FUNCTION_BLOCK JackControl (* Composite Function Block Type *)
  (* Standard: 61499-2 *)
  (* Version 0.0, 4/16/2020, prana, nxtControl GmbH, template *)
  PACKAGE Main;
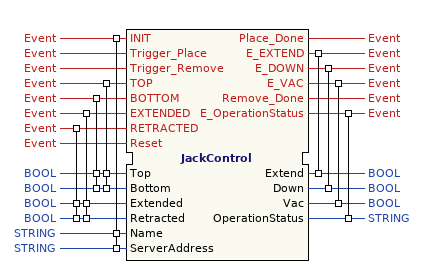
  EVENT_INPUT
    INIT WITH Name, ServerAddress; (* Initialization Request *)
    Trigger_Place;
    Trigger_Remove;
    TOP WITH Top, Bottom; {SET_ATTRIBUTE(Runtime.OPCUA.Access, 2)}
    BOTTOM WITH Bottom, Top; {SET_ATTRIBUTE(Runtime.OPCUA.Access, 2)}
    EXTENDED WITH Extended, Retracted; {SET_ATTRIBUTE(Runtime.OPCUA.Access, 2)}
    RETRACTED WITH Retracted, Extended; {SET_ATTRIBUTE(Runtime.OPCUA.Access, 2)}
    Reset;
  END_EVENT
  EVENT_OUTPUT
    Place_Done;
    E_EXTEND WITH Extend;
    E_DOWN WITH Down;
    E_VAC WITH Vac;
    Remove_Done;
    E_OperationStatus WITH OperationStatus; (* Execution Confirmation *)
  END_EVENT
  VAR_INPUT
    Top : BOOL; {SET_ATTRIBUTE(Runtime.OPCUA.Access, 2)} {SET_ATTRIBUTE(Runtime.OPCUA.WriteTrigger, TOP)}
    Bottom : BOOL; {SET_ATTRIBUTE(Runtime.OPCUA.Access, 2)} {SET_ATTRIBUTE(Runtime.OPCUA.WriteTrigger, BOTTOM)}
    Extended : BOOL; {SET_ATTRIBUTE(Runtime.OPCUA.Access, 2)} {SET_ATTRIBUTE(Runtime.OPCUA.WriteTrigger, EXTENDED)}
    Retracted : BOOL; {SET_ATTRIBUTE(Runtime.OPCUA.Access, 2)} {SET_ATTRIBUTE(Runtime.OPCUA.WriteTrigger, RETRACTED)}
    Name : STRING;
    ServerAddress : STRING;
  END_VAR
  VAR_OUTPUT
    Extend : BOOL; {SET_ATTRIBUTE(Runtime.OPCUA.Access, 2)}
    Down : BOOL; {SET_ATTRIBUTE(Runtime.OPCUA.Access, 2)}
    Vac : BOOL; {SET_ATTRIBUTE(Runtime.OPCUA.Access, 2)}
    OperationStatus : STRING; (* Output event qualifier *)
  END_VAR
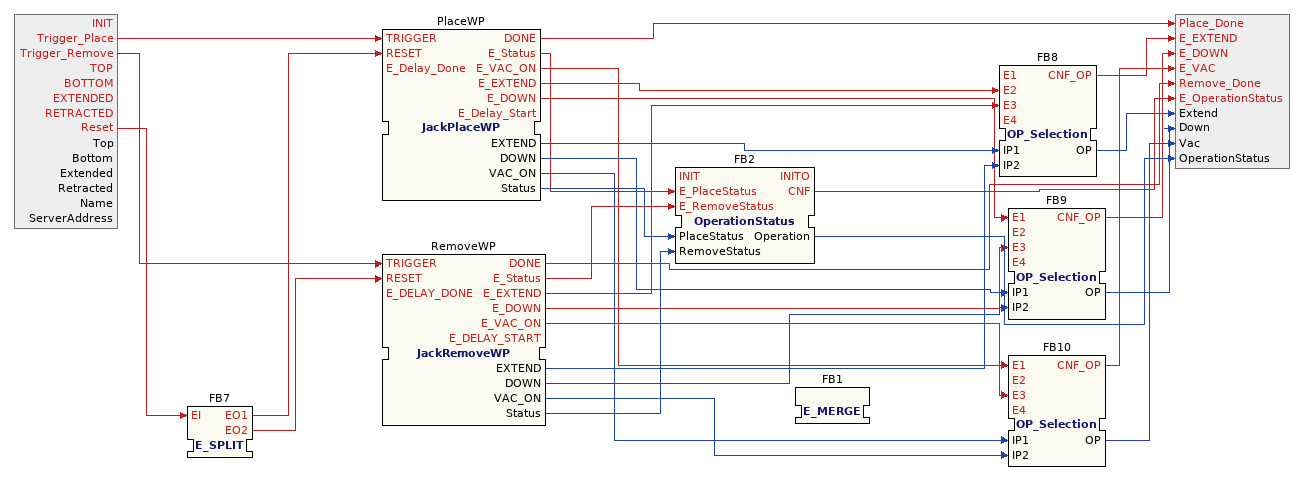
  FBS
    PlaceWP : JackPlaceWP;
    RemoveWP : JackRemoveWP;
    FB7 : E_SPLIT;
    FB8 : OP_Selection;
    FB9 : OP_Selection;
    FB10 : OP_Selection;
    FB1 : E_MERGE;
    FB2 : OperationStatus;
  END_FBS
  EVENT_CONNECTIONS
    Trigger_Place TO PlaceWP.TRIGGER;
    Trigger_Remove TO RemoveWP.TRIGGER;
    Reset TO FB7.EI;
    FB7.EO1 TO PlaceWP.RESET;
    FB7.EO2 TO RemoveWP.RESET;
    FB8.CNF_OP TO E_EXTEND;
    FB9.CNF_OP TO E_DOWN;
    FB10.CNF_OP TO E_VAC;
    RemoveWP.E_VAC_ON TO FB10.E3;
    PlaceWP.E_VAC_ON TO FB10.E1;
    RemoveWP.E_DOWN TO FB9.E3;
    PlaceWP.E_DOWN TO FB9.E1;
    PlaceWP.E_EXTEND TO FB8.E2;
    RemoveWP.E_EXTEND TO FB8.E3;
    PlaceWP.DONE TO Place_Done;
    RemoveWP.DONE TO Remove_Done;
    PlaceWP.E_Status TO FB2.E_PlaceStatus;
    RemoveWP.E_Status TO FB2.E_RemoveStatus;
    FB2.CNF TO E_OperationStatus;
  END_CONNECTIONS
  DATA_CONNECTIONS
    FB8.OP TO Extend;
    FB9.OP TO Down;
    FB10.OP TO Vac;
    RemoveWP.VAC_ON TO FB10.IP2;
    PlaceWP.VAC_ON TO FB10.IP1;
    RemoveWP.DOWN TO FB9.IP2;
    PlaceWP.DOWN TO FB9.IP1;
    RemoveWP.EXTEND TO FB8.IP2;
    PlaceWP.EXTEND TO FB8.IP1;
    FB2.Operation TO OperationStatus;
    PlaceWP.Status TO FB2.PlaceStatus;
    RemoveWP.Status TO FB2.RemoveStatus;
  END_CONNECTIONS
END_FUNCTION_BLOCK
